// TIA Portal V17 export
// export: Created 2024-09-02T12:50:31.4968265Z, ExportSetting WithDefaults, DisplayName Totally Integrated Automation Portal, DisplayVersion V17, DisplayName TIA Portal Openness, DisplayVersion V17, DisplayName TIA Portal Version Control Interface, DisplayVersion V17, DisplayName STEP 7 Professional, DisplayVersion V17, DisplayName STEP 7 Safety, DisplayVersion V17, DisplayName WinCC Professional, DisplayVersion V17
TYPE "UFM_IoDataArray"
TITLE = UFM_IoDataArray
// Type of the mapped input and output fieldbus data to be passed to UFM_Station.
// stored: IsFailsafeCompliant false
   STRUCT
      Values : Array[1..32] of Word;
   END_STRUCT;
END_TYPE
